PROGRAM Background_Time
VAR
	fbTime 		: FB_LocalSystemTime := ( bEnable := TRUE, dwCycle := 1 );
	bValid		: BOOL := FALSE;
	TimeStr		: STRING;
	cSec		: WORD;
	cMil		: WORD;
END_VAR

(* get system time *)
WHILE bValid = FALSE DO
	fbTime(bValid => bValid);	
END_WHILE

fbTime();

TimeStr	:= SYSTEMTIME_TO_STRING(Background_Time.fbTime.systemTime);
cSec	:= fbTime.systemTime.wSecond;
cMil	:= fbTime.systemTime.wMilliseconds;

END_PROGRAM

(* stored: Version 1.1.0.1, ProductVersion 3.1.4024.6
   POU Background_Time: Id {77380658-b361-4e3d-9124-8dca135a14c1}, SpecialFunc None *)
